KUKA KRL program: speedtest2a.src

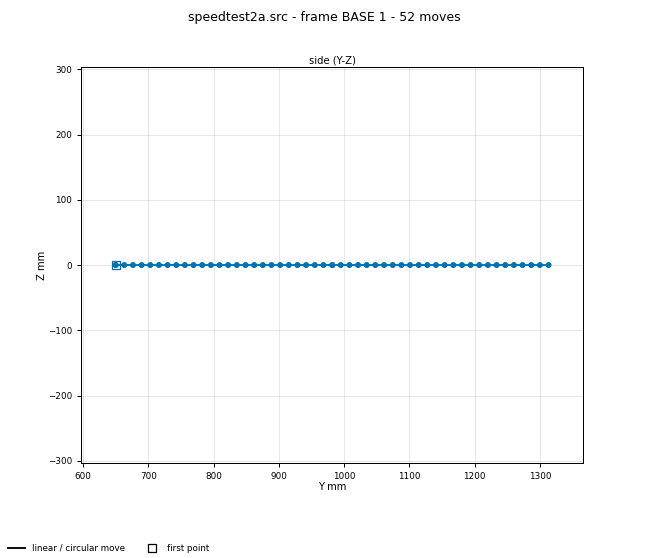
[picture p0: tool path of speedtest2a.src in frame BASE 1, 52 of 53 moves have a stored position in this frame; points joined in program order, loops and branches not executed]
&ACCESS RVEO
&REL 11
&PARAM TEMPLATE = C:\KRC\Roboter\Template\vorgabe
&PARAM EDITMASK = *
DEF variable_helical2( )
;FOLD INI
  ;FOLD BASISTECH INI
    GLOBAL INTERRUPT DECL 3 WHEN $STOPMESS==TRUE DO IR_STOPM ( )
    INTERRUPT ON 3
    BAS (#INITMOV,0 )
  ;ENDFOLD (BASISTECH INI)
 ;FOLD USER INI


    ;Make your modifications here
  ;ENDFOLD (USER INI)
;ENDFOLD (INI)
ACTION(#AXIS_RESET,34,1000,#NOERROR,ERROR_CODE)
;FOLD PTP HOME  Vel= 100 % DEFAULT;%{PE}%MKUKATPBASIS,%CMOVE,%VPTP,%P 1:PTP, 2:HOME, 3:, 5:100, 7:DEFAULT
$BWDSTART = FALSE
PDAT_ACT=PDEFAULT
FDAT_ACT=FHOME
BAS (#PTP_PARAMS,100 )
$H_POS=XHOME
PTP  XHOME
;ENDFOLD
BAS(#TOOL,1)
BAS(#BASE,1)
$VEL_AXIS[1]=100
$VEL_AXIS[2]=100
$VEL_AXIS[3]=100
$VEL_AXIS[4]=100
$VEL_AXIS[5]=100
$VEL_AXIS[6]=100
$VEL_EXTAX[1]=100
$VEL_EXTAX[2]=100

$ACC_AXIS[1]=100
$ACC_AXIS[2]=100
$ACC_AXIS[3]=100
$ACC_AXIS[4]=100
$ACC_AXIS[5]=100
$ACC_AXIS[6]=100
$ACC_EXTAX[1]=100
$ACC_EXTAX[2]=100

LIN {Y     +650.000, X     -154.997, Z       +0.000, A       +0.000, E1       +0.000}
LIN_REL {Y       +13.265, X       +0.000, Z       +0.000, A       +0.000, E3      +0.000, E1       +0.000}
LIN_REL {Y       +13.265, X       +0.000, Z       +0.000, A       +0.000, E3      +0.000, E1       +0.000}
LIN_REL {Y       +13.265, X       +0.000, Z       +0.000, A       +0.000, E3      +0.000, E1       +0.000}
LIN_REL {Y       +13.265, X       +0.000, Z       +0.000, A       +0.000, E3      +0.000, E1       +0.000}
LIN_REL {Y       +13.265, X       +0.000, Z       +0.000, A       +0.000, E3      +0.000, E1       +0.000}
LIN_REL {Y       +13.265, X       +0.000, Z       +0.000, A       +0.000, E3      +0.000, E1       +0.000}
LIN_REL {Y       +13.265, X       +0.000, Z       +0.000, A       +0.000, E3      +0.000, E1       +0.000}
LIN_REL {Y       +13.265, X       +0.000, Z       +0.000, A       +0.000, E3      +0.000, E1       +0.000}
LIN_REL {Y       +13.265, X       +0.000, Z       +0.000, A       +0.000, E3      +0.000, E1       +0.000}
LIN_REL {Y       +13.265, X       +0.000, Z       +0.000, A       +0.000, E3      +0.000, E1       +0.000}
LIN_REL {Y       +13.265, X       +0.000, Z       +0.000, A       +0.000, E3      +0.000, E1       +0.000}
LIN_REL {Y       +13.265, X       +0.000, Z       +0.000, A       +0.000, E3      +0.000, E1       +0.000}
LIN_REL {Y       +13.265, X       +0.000, Z       +0.000, A       +0.000, E3      +0.000, E1       +0.000}
LIN_REL {Y       +13.265, X       +0.000, Z       +0.000, A       +0.000, E3      +0.000, E1       +0.000}
LIN_REL {Y       +13.265, X       +0.000, Z       +0.000, A       +0.000, E3      +0.000, E1       +0.000}
LIN_REL {Y       +13.265, X       +0.000, Z       +0.000, A       +0.000, E3      +0.000, E1       +0.000}
LIN_REL {Y       +13.265, X       +0.000, Z       +0.000, A       +0.000, E3      +0.000, E1       +0.000}
LIN_REL {Y       +13.265, X       +0.000, Z       +0.000, A       +0.000, E3      +0.000, E1       +0.000}
LIN_REL {Y       +13.265, X       +0.000, Z       +0.000, A       +0.000, E3      +0.000, E1       +0.000}
LIN_REL {Y       +13.265, X       +0.000, Z       +0.000, A       +0.000, E3      +0.000, E1       +0.000}
LIN_REL {Y       +13.265, X       +0.000, Z       +0.000, A       +0.000, E3      +0.000, E1       +0.000}
LIN_REL {Y       +13.265, X       +0.000, Z       +0.000, A       +0.000, E3      +0.000, E1       +0.000}
LIN_REL {Y       +13.265, X       +0.000, Z       +0.000, A       +0.000, E3      +0.000, E1       +0.000}
LIN_REL {Y       +13.265, X       +0.000, Z       +0.000, A       +0.000, E3      +0.000, E1       +0.000}
LIN_REL {Y       +13.265, X       +0.000, Z       +0.000, A       +0.000, E3      +0.000, E1       +0.000}
LIN_REL {Y       +13.265, X       +0.000, Z       +0.000, A       +0.000, E3      +0.000, E1       +0.000}
LIN_REL {Y       +13.265, X       +0.000, Z       +0.000, A       +0.000, E3      +0.000, E1       +0.000}
LIN_REL {Y       +13.265, X       +0.000, Z       +0.000, A       +0.000, E3      +0.000, E1       +0.000}
LIN_REL {Y       +13.265, X       +0.000, Z       +0.000, A       +0.000, E3      +0.000, E1       +0.000}
LIN_REL {Y       +13.265, X       +0.000, Z       +0.000, A       +0.000, E3      +0.000, E1       +0.000}
LIN_REL {Y       +13.265, X       +0.000, Z       +0.000, A       +0.000, E3      +0.000, E1       +0.000}
LIN_REL {Y       +13.265, X       +0.000, Z       +0.000, A       +0.000, E3      +0.000, E1       +0.000}
LIN_REL {Y       +13.265, X       +0.000, Z       +0.000, A       +0.000, E3      +0.000, E1       +0.000}
LIN_REL {Y       +13.265, X       +0.000, Z       +0.000, A       +0.000, E3      +0.000, E1       +0.000}
LIN_REL {Y       +13.265, X       +0.000, Z       +0.000, A       +0.000, E3      +0.000, E1       +0.000}
LIN_REL {Y       +13.265, X       +0.000, Z       +0.000, A       +0.000, E3      +0.000, E1       +0.000}
LIN_REL {Y       +13.265, X       +0.000, Z       +0.000, A       +0.000, E3      +0.000, E1       +0.000}
LIN_REL {Y       +13.265, X       +0.000, Z       +0.000, A       +0.000, E3      +0.000, E1       +0.000}
LIN_REL {Y       +13.265, X       +0.000, Z       +0.000, A       +0.000, E3      +0.000, E1       +0.000}
LIN_REL {Y       +13.265, X       +0.000, Z       +0.000, A       +0.000, E3      +0.000, E1       +0.000}
LIN_REL {Y       +13.265, X       +0.000, Z       +0.000, A       +0.000, E3      +0.000, E1       +0.000}
LIN_REL {Y       +13.265, X       +0.000, Z       +0.000, A       +0.000, E3      +0.000, E1       +0.000}
LIN_REL {Y       +13.265, X       +0.000, Z       +0.000, A       +0.000, E3      +0.000, E1       +0.000}
LIN_REL {Y       +13.265, X       +0.000, Z       +0.000, A       +0.000, E3      +0.000, E1       +0.000}
LIN_REL {Y       +13.265, X       +0.000, Z       +0.000, A       +0.000, E3      +0.000, E1       +0.000}
LIN_REL {Y       +13.265, X       +0.000, Z       +0.000, A       +0.000, E3      +0.000, E1       +0.000}
LIN_REL {Y       +13.265, X       +0.000, Z       +0.000, A       +0.000, E3      +0.000, E1       +0.000}
LIN_REL {Y       +13.265, X       +0.000, Z       +0.000, A       +0.000, E3      +0.000, E1       +0.000}
LIN_REL {Y       +13.265, X       +0.000, Z       +0.000, A       +0.000, E3      +0.000, E1       +0.000}
LIN_REL {Y       +13.265, X       +0.000, Z       +0.000, A       +0.000, E3      +0.000, E1       +0.000}

LIN {Y     +650.000, X     -154.997, Z       +0.000, A       +0.000, E1       +0.000}

HALT


END
